// TIA Portal V16 export
// export: Created 2024-12-03T15:41:45.9755271Z, ExportSetting WithReadOnly, DisplayName Totally Integrated Automation Portal, DisplayVersion V16 Update 6, DisplayName TIA Portal Version Control Interface, DisplayVersion V16 Update 2, DisplayName TIA Portal Openness, DisplayVersion V16 Update 6, DisplayName TIA Portal Teamcenter Gateway, DisplayVersion V16, DisplayName SINAMICS Startdrive Advanced, DisplayVersion V16 Update 5, DisplayName SINAMICS Startdrive G130, G150, S120, S150, SINAMICS MV, S210, DisplayVersion V16 Update 5, DisplayName SINAMICS Startdrive G110M, G120, G120C, G120D, G120P, G115D, DisplayVersion V16 Update 5, DisplayName STEP 7 Professional, DisplayVersion V16 Update 6, DisplayName STEP 7 Safety, DisplayVersion V16, DisplayName WinCC Advanced / Unified PC, DisplayVersion V16 Update 6
TYPE "Intersection"
// stored: CreationDate 2021-07-13T07:41:36.2278727Z, InterfaceModifiedDate 2023-07-10T11:57:51.3767682Z, IsConsistent true, LibraryConformanceStatus The object is library-conformant., ModifiedDate 2023-07-10T11:57:51.3767682Z
   STRUCT
      UpstreamIndex : Int;
      DownstreamIndex : Int;
      ReceivePosition : Int;
      SendingPosition : Int;
      ReceiveConveyorIndex : Int;
      SendingConveyorIndex : Int;
      InverseFlowReceiving : Bool;
      InverseFlowSending : Bool;
      ReceiveNoEndSensor : Bool;
      TargetConveyor : Int;
      RequestingConveyor : Int;
      Algin : Struct
         active : Bool;
         speed : Real;
         direction : Bool;
         AlginPosition : Int;   // -1 = down / 1 = up
         conveyorIndex : UInt;   // 1 = conv_1 / 2 = conv_2
         distnace : Real;
      END_STRUCT;
   END_STRUCT;
END_TYPE
